// TIA Portal V19 export
DATA_BLOCK "DB_ExportFlatCtrlRobot1"   // DB72
{ S7_Optimized_Access := 'TRUE' }
// stored: AutoNumber false, IsOnlyStoredInLoadMemory true, MemoryReserve 100
   VAR RETAIN
      FlatnessRecords { S7_SetPoint := 'True'} : Array[0..200] of "stFlatnessCtrlRecord";
   END_VAR
BEGIN
   FlatnessRecords[1].dtlDataTime := DTL#2025-07-23-18:30:25.845572084;
   FlatnessRecords[1].xFlatnessResult := TRUE;
   FlatnessRecords[1].uiStrokePositionDiskA := 237;
   FlatnessRecords[1].uiStrokePositionDiskB := 237;
   FlatnessRecords[1].uiStrokePositionDiskC := 240;
END_DATA_BLOCK
